(* CODESYS project CodeSys-projekti.export

Project tree, tasks and I/O mapping:
  HMI_BO : CDPX, Festo AG & Co. KG, order no. 574410, 574411, 574412, 574413, version 3.5.4.0
  PLC_BO : CDPX, Festo AG & Co. KG, order no. CDPX-X-A-W-4(574410),CDPX-X-A-W-7(574411),CDPX-X-A-S-10(574412),CDPX-X-A-W-13(574413), version 3.5.7.25
    application Application
      libraries: Util, 3.5.0.0 (System); CmpApp, 3.5.4.0 (System); CmpEventMgr, 3.5.4.0 (System); CmpIecTask, 3.5.2.0 (System); Component Manager, 3.5.5.0 (System); Standard, 3.5.17.0 (System)
      task Task20ms (cyclic, interval t#20ms, priority 10) calls PLC_PRG
      Data types/
      Global Variables/
        global variables Global_variables
        global variables Variablen_Konfiguration
      POUs/
        function block FBD_Analog_motor_control [FBD]
        function block FBD_Auto_Conveyor_valve [FBD]
        function block FBD_Auto_output_control [FBD]
        function block FBD_Auto_pump_on [FBD]
        function block LD_Automaattitila [LD]
        function block LD_Manuaali_logiikka [LD]
        function block Manuaalitila_setpiiri [LD]
        program PLC_PRG [LD]
        function block ST_Data_manipulation [ST]
      SymbolConfigObject
    CDPX_EA_V1 : CDPX-EA-V1, Festo AG & Co. KG, order no. 575300, version 3.5.7.1
        unmapped channels: Inputs, Outputs, Value, OverFlow, UnderFlow, ZeroDetect, Value, OverFlow, UnderFlow, ZeroDetect, CntTrgEncLd, Mode, ClockPrescaler, InputPrescaler, ZeroSearchEnable, ClearCounter, CounterStyle, ClearFlags, MachineZeroEnable, MachinePol, EncZeroEnable, EncPol, InpEdge, GatePol, CntTrgEncLd, Mode, ClockPrescaler, InputPrescaler, ZeroSearchEnable, ClearCounter, CounterStyle, ClearFlags, MachineZeroEnable, MachinePol, EncZeroEnable, EncPol, InpEdge, GatePol, Channel 1, Channel 2,
          Channel 3, Channel 4, Comp, Channel 1, Channel 2, Channel 3, Channel 4
      Digital inputs
          unmapped channels: Inputs
      Digital outputs
          unmapped channels: Outputs
      Counter/Encoder
          unmapped channels: Value, OverFlow, UnderFlow, ZeroDetect, Value, OverFlow, UnderFlow, ZeroDetect, CntTrgEncLd, Mode, ClockPrescaler, InputPrescaler, ZeroSearchEnable, ClearCounter, CounterStyle, ClearFlags, MachineZeroEnable, MachinePol, EncZeroEnable, EncPol, InpEdge, GatePol, CntTrgEncLd, Mode, ClockPrescaler, InputPrescaler, ZeroSearchEnable, ClearCounter, CounterStyle, ClearFlags, MachineZeroEnable, MachinePol, EncZeroEnable, EncPol, InpEdge, GatePol
      Analog inputs
          unmapped channels: Channel 1, Channel 2, Channel 3, Channel 4, Comp
      Analog outputs
          unmapped channels: Channel 1, Channel 2, Channel 3, Channel 4
*)

// PLC_BO/Application/Global Variables/Global_variables

VAR_GLOBAL
    // ======================================================
    // 1. HMI-painonapit ja ohjausarvot
    // ======================================================
    S1 : BOOL;    (* Manuaalitila päälle, HMI *)
    S2 : BOOL;    (* Automaattitila päälle, HMI *)
    S3 : BOOL;    (* Nollaus, HMI *)
    S4 : BOOL;    (* PL2 pumppu päälle, HMI *)
    S5 : BOOL;    (* MA1 ja MA2 kuljettimet päälle, HMI *)
    S6 : BOOL;    (* Pullotusventtiili päälle, HMI *)
    S7 : BOOL;    (* Lajittelija kuljetin päälle, HMI *)
    S8 : BOOL;    (* Automaattitila START, HMI *)
    S9 : BOOL;    (* Automaattitila STOP/RESUME, HMI *)

    HMI_Prosentti : REAL;        // 0.0–100.0 HMI:stä lähtevä arvo
    HMI_PL1_ON : BOOL;           // HMI syöttö PL1 pumppu ON/OFF
    HMI_valve_timer : TIME;      // HMI Valve ON timer
    HMI_fill : INT;              // Täyttömäärä (ml)

	HMI_4B3_alarm:BOOL;			// HMI alarm for Empty tank
    // ======================================================
    // 2. Fyysiset digitaaliset tulot (I/O)
    // ======================================================
    _4B1 AT %IX0.0 : BOOL;   (* B402 reached, VE2 tasokytkin *)
    _4B2 AT %IX0.1 : BOOL;   (* B401 top, VE1 yläraja *)
    _4B3 AT %IX0.2 : BOOL;   (* B401 bottom, VE1 alaraja *)
    _4B4 AT %IX0.3 : BOOL;   (* Pullo kuljettimen alussa *)
    _4B5 AT %IX0.4 : BOOL;   (* Pullo täyttöpisteessä *)
    _4B6 AT %IX0.5 : BOOL;   (* Pullo kuljettimen lopussa *)
    xOverflow AT %IX0.7 : BOOL; (* Kellukekytkinten ylivuoto *)
    EmStop AT %IX1.5 : BOOL;    (* Hätäseis *)
    I6com_PA_FREE AT %IX1.6 : BOOL; (* PA asema vapaa *)
    I7com_Belt_FREE AT %IX1.7 : BOOL; (* MPS kuljetin vapaa *)

    // ======================================================
    // 3. Fyysiset digitaaliset lähdöt (I/O)
    // ======================================================
    _4M1 AT %QX0.0 : BOOL;   (* PL1 pumppu ON *)
    _4M2 AT %QX0.1 : BOOL;   (* Pullotusventtiili ON *)
    _4M3 AT %QX0.2 : BOOL;   (* Kuljettimet ON *)
    _4M4 AT %QX0.3 : BOOL;   (* Lajittelija ON *)
    MA5 AT %QX0.4 : BOOL;    (* PL2 pumppu ON *)
    Q4com_PA_Ready AT %QX1.2 : BOOL; (* PA asema valmis *)
    Q6com_Belt_Rdy AT %QX1.3 : BOOL; (* Kuljetin valmis *)

    // ======================================================
    // 4. Analogiset arvot (I/O)
    // ======================================================
    _4CO1 AT %QD7 : DINT;    (* Stellgröße Y / ohjausarvo PL1 *)
    _4CO2 AT %QD8 : DINT;    (* Sollwert SP / asetusarvo *)
    _4PV1 AT %ID5 : DINT;    (* Istwert X / prosessiarvo *)

    // ======================================================
    // 5. Prosessin ohjausmuuttujat
    // ======================================================
	Fill_Start : BOOL;           // Täytön aloitus
    Fill_ready : BOOL;           // Täyttö valmis
    Fill_ready_timer : BOOL;     // Viive valmis (timer)
    Auto_PL1_ON : BOOL;          // Automaattinen PL1 ohjaus
	Auto_filling_valve : BOOL;	 // Automaattitilan täyttöventtiili ohjaus
	Auto_conveyor_motor : BOOL;	 // Automaattitilan Kuljetin moottorin ohjaus
	Auto_seperator : BOOL;		 // Automaattitilan lajittelija ohjaus
    Automaattitila_Paalle : BOOL;// Automaattitila aktiivinen
    Manuaalitila_Paalle : BOOL;  // Manuaalitila aktiivinen
	bottles_on_conveyor : BOOL; // TRUE, jos CTUD_0.CV > 0 (pulloja linjalla)
	Empty_tank_stop : BOOL; 	// sammutusbitti
	
    // ======================================================
    // 6. Anturin laskennalliset arvot
    // ======================================================
    Tilavuus_ml : REAL;          // Tilavuus VE2 millilitroina
    Korkeus_mm : REAL;           // Veden korkeus VE2 millimetreinä

    // ======================================================
    // 7. Mahdolliset lisämuuttujat (kommentoituna)
    // ======================================================
    // SR : BOOL;    (* Status-signaali, ei käytössä nyt *)
    // Alarm : BOOL; (* Hälytys, ei käytössä nyt *)
    // I6com_PA_FREE : BOOL; (* Looginen kopio, poistettu duplikaattina *)
    // I7com_Belt_FREE : BOOL; (* Looginen kopio, poistettu duplikaattina *)
END_VAR

// PLC_BO/Application/Global Variables/Variablen_Konfiguration
VAR_CONFIG
END_VAR

// PLC_BO/Application/POUs/PLC_PRG
PROGRAM PLC_PRG
VAR
	ST_Data_manipulation_0: ST_Data_manipulation;
	
	Manuaalitila_setpiiri : Manuaalitila_setpiiri;
	LD_Automaattitila_0: LD_Automaattitila;
	
	FBD_Auto_Conveyor_valve: FBD_Auto_Conveyor_valve;
	FBD_Auto_pump_on_0: FBD_Auto_pump_on;
	FBD_Analog_motor_control_0: FBD_Analog_motor_control;
	LD_Manuaali_logiikka_0: LD_Manuaali_logiikka;
	
	
	
	FBD_Auto_output_control_0: FBD_Auto_output_control;
END_VAR
VAR // added by the converter: edge detectors and wires of the graphical bodies
    _w1, _w2, _w3 : BOOL;
END_VAR

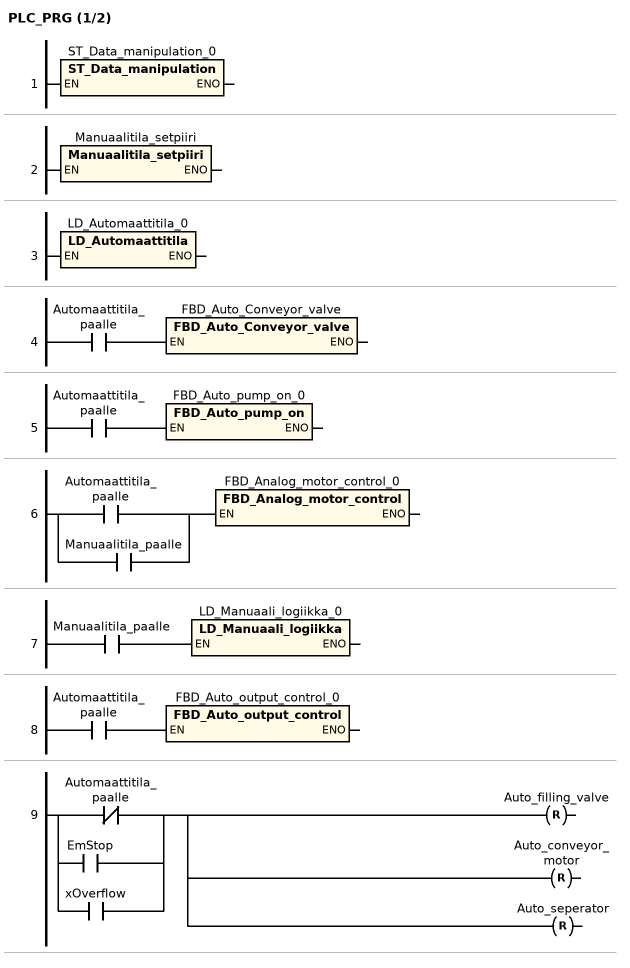
// NETWORK 1
ST_Data_manipulation_0(); // ST_Data_manipulation

// NETWORK 2
Manuaalitila_setpiiri();

// NETWORK 3
LD_Automaattitila_0(); // LD_Automaattitila

// NETWORK 4
IF Automaattitila_paalle THEN FBD_Auto_Conveyor_valve(); END_IF

// NETWORK 5
IF Automaattitila_paalle THEN
    FBD_Auto_pump_on_0(); // FBD_Auto_pump_on
END_IF

// NETWORK 6
IF Automaattitila_paalle OR Manuaalitila_paalle THEN
    FBD_Analog_motor_control_0(); // FBD_Analog_motor_control
END_IF

// NETWORK 7
IF Manuaalitila_paalle THEN
    LD_Manuaali_logiikka_0(); // LD_Manuaali_logiikka
END_IF

// NETWORK 8
IF Automaattitila_paalle THEN
    FBD_Auto_output_control_0(); // FBD_Auto_output_control
END_IF

// NETWORK 9
_w1 := NOT Automaattitila_paalle OR EmStop OR xOverflow;
Auto_filling_valve R= _w1;
Auto_conveyor_motor R= _w1;
Auto_seperator R= _w1;

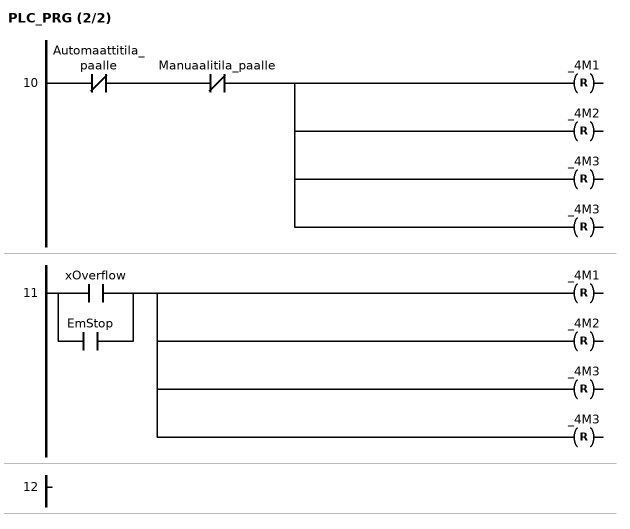
// NETWORK 10
_w2 := NOT Automaattitila_paalle AND NOT Manuaalitila_paalle;
_4M1 R= _w2;
_4M2 R= _w2;
_4M3 R= _w2;
_4M3 R= _w2;

// NETWORK 11
_w3 := xOverflow OR EmStop;
_4M1 R= _w3;
_4M2 R= _w3;
_4M3 R= _w3;
_4M3 R= _w3;

// NETWORK 12

END_PROGRAM

// PLC_BO/Application/POUs/ST_Data_manipulation
FUNCTION_BLOCK ST_Data_manipulation
VAR CONSTANT
    MinArvo : DINT := 5000;       // Anturin arvo pohjalla
    MaxArvo : DINT := 9630000;    // Anturin arvo täydessä säiliössä
    TilavuusMax : REAL := 3390.0; // Säiliön tilavuus ml
    KorkeusMax : REAL := 220.0;   // Säiliön korkeus mm
END_VAR
VAR_INPUT
END_VAR
VAR_OUTPUT
END_VAR
VAR
    Snapshot : REAL;              // Tallennettu tilavuus
    RajoitettuArvo : DINT;        // Anturin arvo rajattuna min-max välille
END_VAR

// Säiliö tyhjenee sammuttaa automaatin *ota pois jossei toimi*
VAR
    // --- Parametrit (säädettävissä) ---
    EmptyThreshold_ml : REAL := 10.0;       // "Tyhjä" jos Tilavuus_ml <= 10 ml
    NotEmptyThreshold_ml : REAL := 20.0;    // "Ei-tyhjä" jos Tilavuus_ml >= 20 ml (hystereesi)
    WaterPresenceThreshold_ml : REAL := 50.0; // "Vettä on ollut" jos joskus >= 50 ml

    // --- Sisäiset tilat ---
    had_water_since_start : BOOL := FALSE;  // latchettu tieto: onko vettä ollut ajon aikana
    empty_state : BOOL := FALSE;            // hysteresis-pohjainen tyhjyyden tila

    // --- Ajastimet ---
    tEmpty5s : TON;                         // 5 s varmistus kun empty_state = TRUE
    // (Ei monofloppia, koska teemme syklipulssin R_TRIG:llä vakiona)

    // --- Pulssin generointi ---
    rTrig_EmptyOk : R_TRIG;                 // Reunanhavaitseminen (nouseva reuna)

    // --- Välisignaalit ---
    allow_stop : BOOL;                      // pysäytys sallittu (ei pulloja linjalla)
    timer_in : BOOL;                        // TON:lle syöttö
END_VAR

// *** Resetointi napilla S3 ***
IF S3 THEN
    HMI_valve_timer := T#0MS;
    HMI_fill := 0;
    Snapshot := 0;
END_IF;

// *** Rajaukset automaattiajon käynnistyspulssilla S8 ***
IF S8 THEN
    // Rajataan HMI_fill välille 500–3000 ml
    IF HMI_fill <= 500 THEN
        HMI_fill := 500;
    ELSIF HMI_fill > 3000 THEN
        HMI_fill := 3000;
    END_IF;

    // Rajataan HMI_valve_timer välille 0–2000 ms
    IF HMI_valve_timer < T#0MS THEN
        HMI_valve_timer := T#0MS;
    ELSIF HMI_valve_timer > T#2000MS THEN
        HMI_valve_timer := T#2000MS;
    END_IF;
END_IF;

// *** Snapshot otetaan S8 painikkeen painalluksesta ***
IF S8 THEN
    Snapshot := Tilavuus_ml + HMI_fill;
END_IF;

// *** Täytön aloitus ***
IF (HMI_fill >= 500) AND Automaattitila_paalle THEN
    Fill_start := TRUE;
ELSE
    Fill_start := FALSE;
END_IF;

// *** Vertailu nykyiseen tilavuuteen ***
IF Tilavuus_ml >= Snapshot THEN
    Fill_ready := TRUE;
ELSE
    Fill_ready := FALSE;
END_IF;

// *** Rajaus anturin arvolle ***
IF _4PV1 < MinArvo THEN
    RajoitettuArvo := MinArvo;
ELSIF _4PV1 > MaxArvo THEN
    RajoitettuArvo := MaxArvo;
ELSE
    RajoitettuArvo := _4PV1;
END_IF;

// *** Skaalaus tilavuudeksi ja korkeudeksi ***
Tilavuus_ml := ((TO_REAL(RajoitettuArvo) - TO_REAL(MinArvo)) * TilavuusMax) / (TO_REAL(MaxArvo) - TO_REAL(MinArvo));
Korkeus_mm := ((TO_REAL(RajoitettuArvo) - TO_REAL(MinArvo)) * KorkeusMax) / (TO_REAL(MaxArvo) - TO_REAL(MinArvo));

// VE1 TANK empty HMI alarm anturin kääntö
IF _4B3=1
	THEN
	HMI_4B3_alarm:=0;
	ELSE
		HMI_4B3_alarm:=1;
END_IF


// --- Päivitetään "säiliössä on ollut vettä" -latch ---
// Kun Tilavuus_ml ylittää veden läsnäolon kynnyksen edes kerran, muistetaan se.
IF Tilavuus_ml >= WaterPresenceThreshold_ml THEN
    had_water_since_start := TRUE;
END_IF;

// --- Resetointi S3:lla palauttaa ajotilanteen ---
// Ei käytetä latcheja hälyn pitämiseen, mutta tämä nollaa muistia "veden ollut" -seurannasta tarvittaessa.
IF S3 THEN
    had_water_since_start := FALSE;
    empty_state := FALSE; // aloita neutraalista tilasta
END_IF;

// ---- AUTOMAATIN SAMMUTUS VEDEN LOPPUESSA	
	// --- Hysteresis: empty_state muodostus ---
	// Anturin heittelyn takia käytetään ala- ja ylärajaa.
	// - Jos tällä hetkellä tyhjä, pysytään tyhjänä kunnes ylitetään NotEmptyThreshold_ml.
	// - Jos ei tyhjä, siirrytään tyhjäksi kun alitetaan EmptyThreshold_ml.
	IF empty_state THEN
		// Tyhjä-tilassa poistutaan vain jos ollaan selvästi ei-tyhjiä
		IF Tilavuus_ml >= NotEmptyThreshold_ml THEN
			empty_state := FALSE;
		END_IF;
	ELSE
		// Ei-tyhjä-tilassa mennään tyhjäksi vasta kun alitetaan tyhjän kynnys
		IF Tilavuus_ml <= EmptyThreshold_ml THEN
			empty_state := TRUE;
		END_IF;
	END_IF;
	
	// --- Stopin esto jos pullot kuljettimella (inhibit) ---
	allow_stop := NOT bottles_on_conveyor;
	
	// --- 5 s varmistusajastin ---
	// Ajastin käy vain, jos: (1) ollaan tyhjänä hysteresis-logiikan mukaan,
	// (2) säiliössä on ollut vettä vähintään kerran ajon aikana,
	// (3) stoppi on sallittu (ei pulloja kuljettimella).
	timer_in := empty_state AND had_water_since_start AND allow_stop;
	tEmpty5s(IN := timer_in, PT := T#5S);
	
	// --- Pulssin generointi, kun 5 s ehto täyttyy ---
	// Käytetään R_TRIG:ä tEmpty5s.Q:n nousevaan reunaan → yksi PLC-sykli pulssi.
	rTrig_EmptyOk(CLK := tEmpty5s.Q);
	
	// --- Ulostulot (pulssi) ---
	// Tuota yksi-syklinen pulssi pysäytykseen ja pudota automaattitila pois samassa syklissä.
	IF rTrig_EmptyOk.Q THEN
		Empty_tank_stop := TRUE;         // pulssi
		Automaattitila_paalle := FALSE;  // pakota automaatti pois
	ELSE
		Empty_tank_stop := FALSE;
	END_IF;

END_FUNCTION_BLOCK

// PLC_BO/Application/POUs/Manuaalitila_setpiiri
FUNCTION_BLOCK Manuaalitila_setpiiri
VAR
    RS_0 : RS; // Kiikku manuaalitilan hallintaan
END_VAR

// Kommentit:
// - RESET = EmStop OR S3 (nollaus).

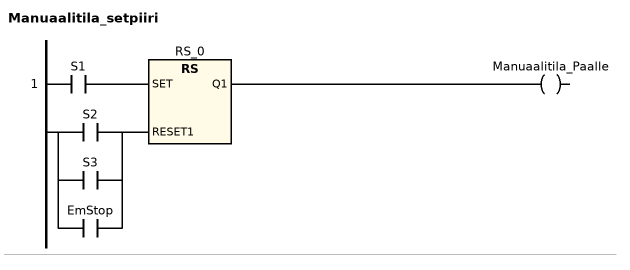
// NETWORK 1
RS_0(SET := S1, RESET1 := S2 OR S3 OR EmStop); // RS
Manuaalitila_Paalle := RS_0.Q1;

END_FUNCTION_BLOCK

// PLC_BO/Application/POUs/LD_Automaattitila
FUNCTION_BLOCK LD_Automaattitila
VAR_INPUT
END_VAR
VAR_OUTPUT
END_VAR
VAR
		// Automaattitila_Paalle
		M1: RS;
END_VAR

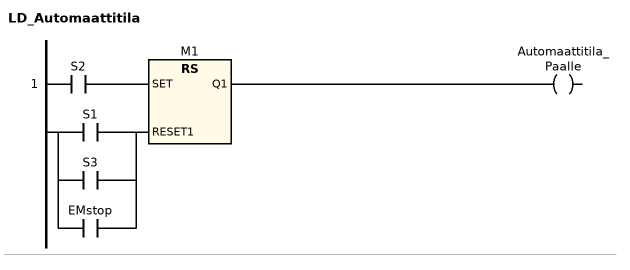
// NETWORK 1
M1(SET := S2, RESET1 := S1 OR S3 OR EMstop); // RS
Automaattitila_Paalle := M1.Q1;

END_FUNCTION_BLOCK

// PLC_BO/Application/POUs/FBD_Auto_Conveyor_valve

FUNCTION_BLOCK FBD_Auto_Conveyor_valve
VAR
    // --- Kiikut ---
    RS_0 : RS;                // Järjestelmä valmis automaattitilassa (SET = Automaattitila, RESET = virheet)
    RS_1 : RS;                // Kuljetin ohjaus (SET = RS_0 & pulloja linjalla, RESET = täyttö, loppupiste, tyhjä linja)

    // --- Ajastimet ---
    TP_1 : TP;                // Venttiilin ohjaus (pulssi HMI_valve_timer-ajaksi, kun pullo saapuu _4B5)
    TP_0 : TP;                // Lajittelijan ohjaus (pulssi 500 ms, kun pullo poistuu _4B5)
    TOF_1 : TOF;              // Jumi-ajastin (pysäyttää ohjelman, jos anturit eivät aktivoidu 30 s)

    // --- Laskuri ---
    CTUD_0 : CTUD;            // Pullojen laskenta (CU = _4B4, CD = _4B6, CV > 0 = pulloja linjalla)

    // --- Reunatunnistukset ---
    R_TRIG_0 : R_TRIG;        // Nousureuna _4B4 (lisää pullo laskuriin)
    F_TRIG_0 : F_TRIG;       // Nousureuna _4B6 (vähentää pullo laskurista)
    R_TRIG_1 : R_TRIG;        // Nousureuna _4B5 (käynnistää TP_1 venttiilin ohjaukseen)
    F_TRIG_1 : F_TRIG;        // Laskeva reuna _4B5 (käynnistää TP_0 lajittelijan pulssin)
	
    // --- Tilabitit ---
    Reset_bit : BOOL;         // Manuaalinen reset (nollaa RS_0 ja RS_1)
    Pause : BOOL;             // Kuljetin pysäytetään täytön ajaksi (TP_1.Q)
    Timer_stop : BOOL;        // Jumi-ajastimen Q (pysäyttää ohjelman)
    Pause_for_load : BOOL;    // Kuljetin pysäytetään latauksen ajaksi (CTUD_0:n Q)
    
	
	// S9 resume
	F_TRIG_2: F_TRIG;
END_VAR
VAR // added by the converter: edge detectors and wires of the graphical bodies
    _w1 : BOOL;
END_VAR

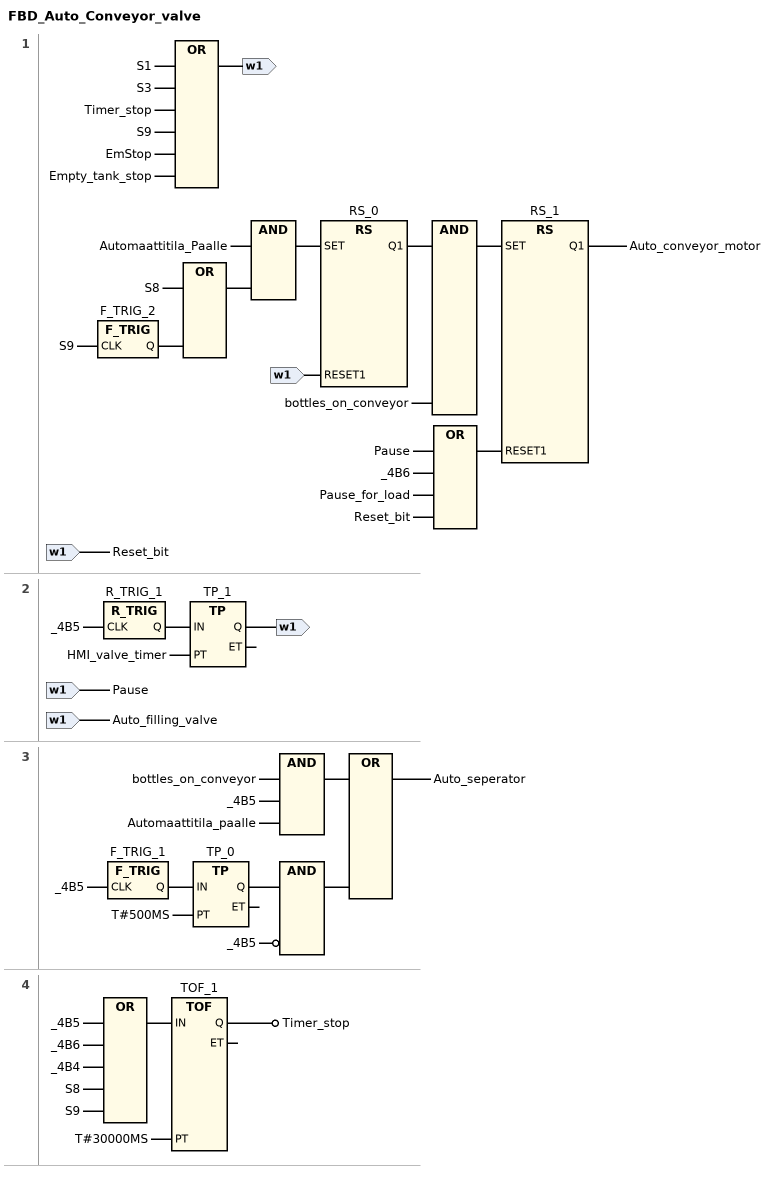
// NETWORK 1
_w1 := S1 OR S3 OR Timer_stop OR S9 OR EmStop OR Empty_tank_stop;
F_TRIG_2(CLK := S9); // F_TRIG
RS_0(SET := Automaattitila_Paalle AND (S8 OR F_TRIG_2.Q), RESET1 := _w1); // RS
RS_1(SET := RS_0.Q1 AND bottles_on_conveyor, RESET1 := Pause OR _4B6 OR Pause_for_load OR Reset_bit); // RS
Auto_conveyor_motor := RS_1.Q1;
Reset_bit := _w1;

// NETWORK 2
R_TRIG_1(CLK := _4B5); // R_TRIG
TP_1(IN := R_TRIG_1.Q, PT := HMI_valve_timer); // TP
Pause := TP_1.Q;
Auto_filling_valve := TP_1.Q;

// NETWORK 3
F_TRIG_1(CLK := _4B5); // F_TRIG
TP_0(IN := F_TRIG_1.Q, PT := T#500MS); // TP
Auto_seperator := bottles_on_conveyor AND _4B5 AND Automaattitila_paalle OR TP_0.Q AND NOT _4B5;

// NETWORK 4
TOF_1(IN := _4B5 OR _4B6 OR _4B4 OR S8 OR S9, PT := T#30000MS); // TOF
Timer_stop := NOT TOF_1.Q;

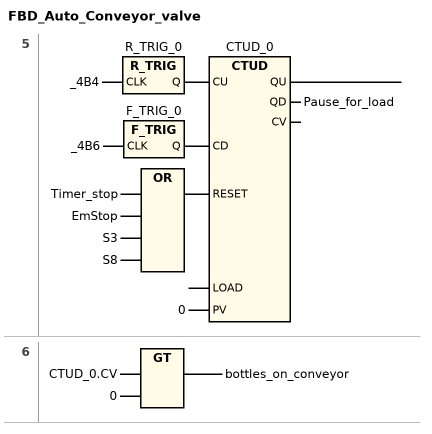
// NETWORK 5
R_TRIG_0(CLK := _4B4); // R_TRIG
F_TRIG_0(CLK := _4B6); // F_TRIG
CTUD_0(
    CU := R_TRIG_0.Q,
    CD := F_TRIG_0.Q,
    RESET := Timer_stop OR EmStop OR S3 OR S8,
    PV := 0,
    QD => Pause_for_load); // CTUD

// NETWORK 6
bottles_on_conveyor := CTUD_0.CV > 0;

END_FUNCTION_BLOCK

// PLC_BO/Application/POUs/FBD_Auto_pump_on

FUNCTION_BLOCK FBD_Auto_pump_on
VAR_INPUT
    // Ei erillisiä syötteitä, ohjaus tulee globaaleista muuttujista
END_VAR
VAR_OUTPUT
    // Auto_PL1_ON ohjaa pumppua automaattitilassa
END_VAR
VAR
    SR_0 : 		SR;    // Kiikku täytön aloitukselle
    RS_1 : 		RS;    // Kiikku pumpun ohjaukselle (RESET prioriteetti)
    TON_0 : 	TON;  // Ajastin roiskeiden suodatukseen
    M7 : TIME := T#1000MS; // Viive roiskeiden poistoon
END_VAR

// Kommentit:
// - TON_0 aktivoituu, kun Fill_ready = TRUE ja automaattitila päällä.
// - Fill_ready_timer = TRUE vasta viiveen jälkeen → estää roiskeiden aiheuttaman virheellisen täyttövalmiuden.
// - RS_1 ohjaa Auto_PL1_ON: SET = Fill_Start, RESET = EmStop OR Fill_ready.
// - Turvallisuus: EmStop katkaisee pumpun välittömästi.

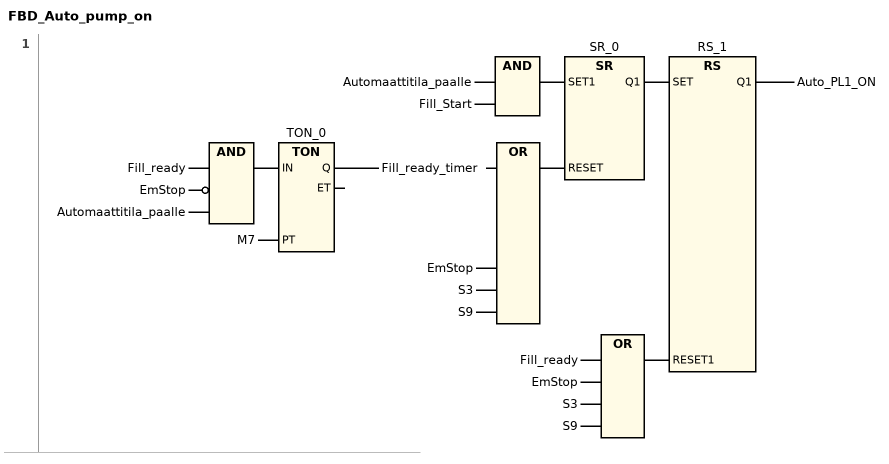
// NETWORK 1
TON_0(IN := Fill_ready AND NOT EmStop AND Automaattitila_paalle, PT := M7); // TON
Fill_ready_timer := TON_0.Q;
SR_0(SET1 := Automaattitila_paalle AND Fill_Start, RESET := TON_0.Q OR EmStop OR S3 OR S9); // SR
RS_1(SET := SR_0.Q1, RESET1 := Fill_ready OR EmStop OR S3 OR S9); // RS
Auto_PL1_ON := RS_1.Q1;

END_FUNCTION_BLOCK

// PLC_BO/Application/POUs/FBD_Analog_motor_control
FUNCTION_BLOCK FBD_Analog_motor_control
VAR_INPUT
    // Ei syötteitä tässä lohkossa, ohjaus tulee globaaleista muuttujista
END_VAR
VAR_OUTPUT
    // Ei erillisiä lähtöjä, ohjaus menee analogiseen kanavaan
END_VAR
VAR
    AnalogOutputChannel : DINT; // Skaalattu ohjausarvo pumpulle (0–10000)
END_VAR

// Kommentit:
// - Skaalaa HMI_Prosentti (0–100 %) analogiseksi ohjaukseksi (0–10000).
// - Valitsee ohjauslähteen: manuaalitila, automaattitila tai HMI_PL1_ON.
// - Käyttää LIMIT-lohkoa varmistamaan, että arvo pysyy 0–10000.
// - Turvallisuus: lisää ehto EmStop → AnalogOutputChannel = 0.

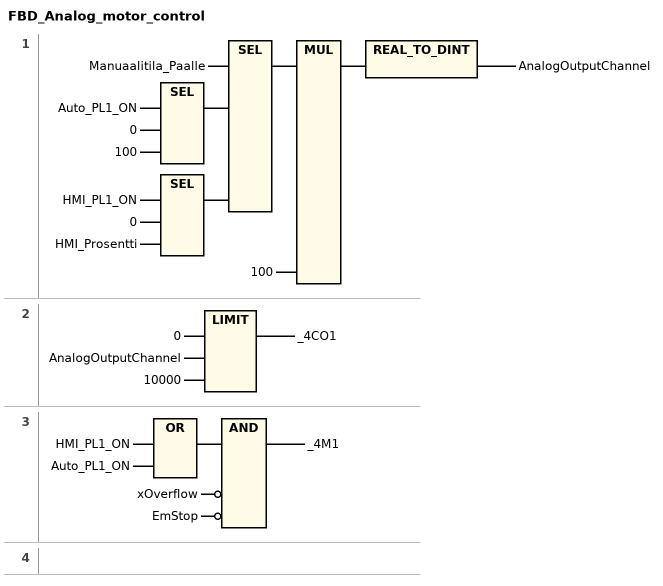
// NETWORK 1
AnalogOutputChannel := REAL_TO_DINT(SEL(Manuaalitila_Paalle, SEL(Auto_PL1_ON, 0, 100), SEL(HMI_PL1_ON, 0, HMI_Prosentti)) * 100);

// NETWORK 2
_4CO1 := LIMIT(0, AnalogOutputChannel, 10000);

// NETWORK 3
_4M1 := (HMI_PL1_ON OR Auto_PL1_ON) AND NOT xOverflow AND NOT EmStop;

// NETWORK 4

END_FUNCTION_BLOCK

// PLC_BO/Application/POUs/LD_Manuaali_logiikka

FUNCTION_BLOCK LD_Manuaali_logiikka
VAR_INPUT
    // Ei erillisiä syötteitä, ohjaus tulee globaaleista muuttujista
END_VAR
VAR_OUTPUT
    // Ohjaa lähdöt manuaalitilassa
END_VAR
VAR
END_VAR

// Kommentit:
// - AND-lohkot ohjaavat lähdöt (venttiili, pumput, kuljettimet) manuaalitilassa.
// - Ehdot: Manuaalitila_Paalle AND HMI-painonappi AND NOT EmStop.
// - EmStop negatoituna (valkoinen pallo) → katkaisee lähdöt välittömästi.

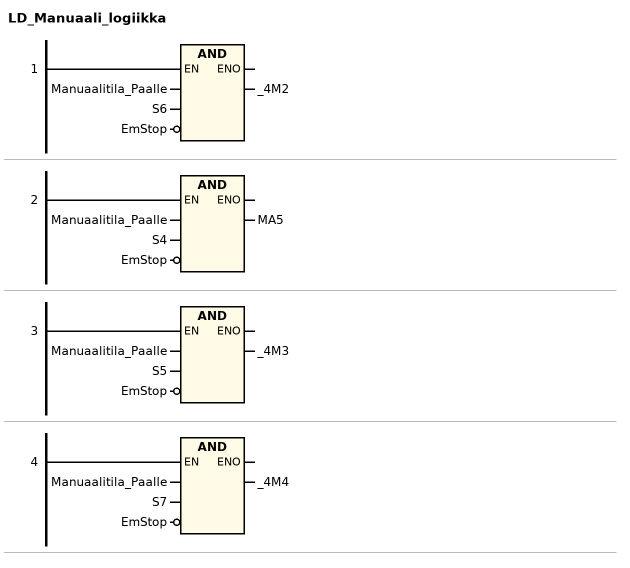
// NETWORK 1
_4M2 := Manuaalitila_Paalle AND S6 AND NOT EmStop;

// NETWORK 2
MA5 := Manuaalitila_Paalle AND S4 AND NOT EmStop;

// NETWORK 3
_4M3 := Manuaalitila_Paalle AND S5 AND NOT EmStop;

// NETWORK 4
_4M4 := Manuaalitila_Paalle AND S7 AND NOT EmStop;

END_FUNCTION_BLOCK

// PLC_BO/Application/POUs/FBD_Auto_output_control
FUNCTION_BLOCK FBD_Auto_output_control
VAR_INPUT
END_VAR
VAR_OUTPUT
END_VAR
VAR
END_VAR

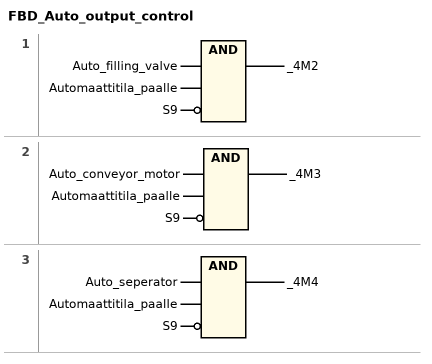
// NETWORK 1
_4M2 := Auto_filling_valve AND Automaattitila_paalle AND NOT S9;

// NETWORK 2
_4M3 := Auto_conveyor_motor AND Automaattitila_paalle AND NOT S9;

// NETWORK 3
_4M4 := Auto_seperator AND Automaattitila_paalle AND NOT S9;

END_FUNCTION_BLOCK
